// TIA Portal V15.1 export
// export: Created 2024-06-21T08:41:24.2160416Z, ExportSetting WithDefaults, DisplayName Totally Integrated Automation Portal, DisplayVersion V15.1 Update 5, DisplayName TIA Portal Openness, DisplayVersion V15.1 Update 5, DisplayName SINAMICS Startdrive Advanced, DisplayVersion V15.1, DisplayName G130, G150, S120, S150, SINAMICS MV, S210, DisplayVersion V15.1, DisplayName G110M, G120, G120C, G120D, G120P, DisplayVersion V15.1, DisplayName STEP 7 Professional, DisplayVersion V15.1 Update 5, DisplayName STEP 7 Safety, DisplayVersion V15.1, DisplayName WinCC Professional, DisplayVersion V15.1 Update 5, DisplayName SIMATIC Visualization Architect, DisplayVersion V15.1
FUNCTION "209210NCB02TagSequence" : Void   // FC341, FBD
TITLE = 209210NCB02TagSequence
{ S7_Optimized_Access := 'TRUE' }
AUTHOR : CSTAAL
VERSION : 0.1
// stored: AutoNumber false, IsIECCheckEnabled false, SetENOAutomatically False, UDAEnableTagReadback false
   VAR_OUTPUT
      O_AlarmA : Bool;   // Alarm A
      O_AlarmB : Bool;   // Alarm B
      O_AlarmC : Bool;   // Alarm C
      O_AlarmD : Bool;   // Alarm D
      O_AlarmABCondition : Bool;   // Alarms resetable
      H_IAnim : Word;   // Icon Animation
   END_VAR
BEGIN

REGION Network 1: **** 1 - Inputs **** HMI Commands
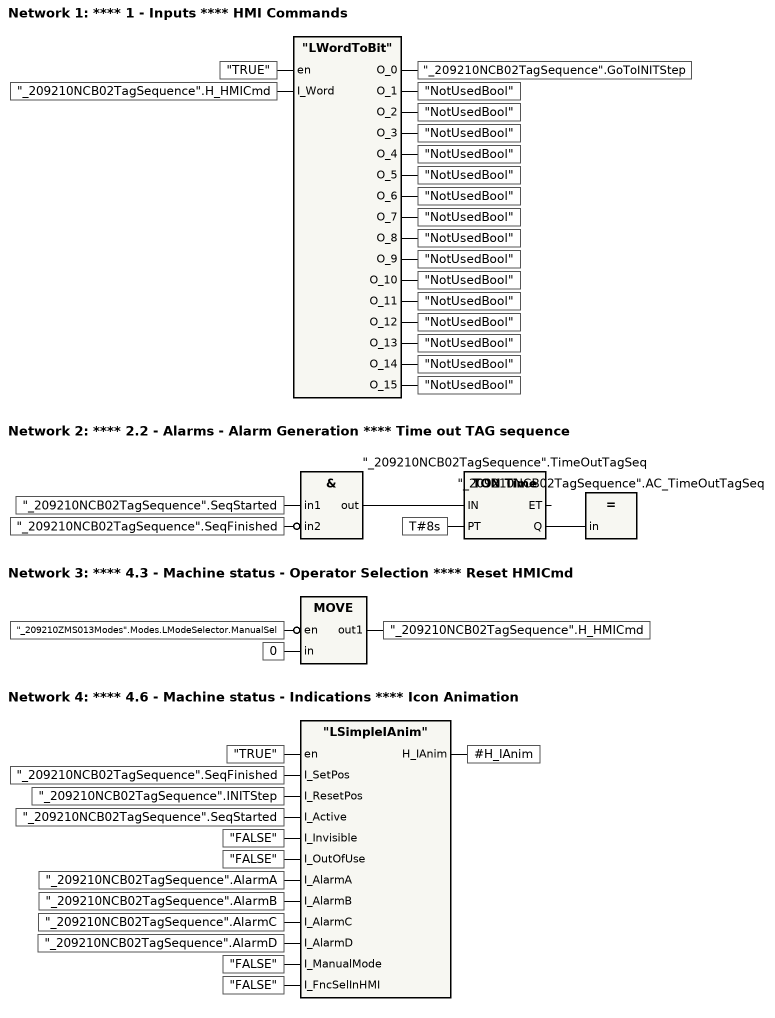
   IF "TRUE" THEN
       "LWordToBit"(I_Word := "_209210NCB02TagSequence".H_HMICmd,
                    O_0 => "_209210NCB02TagSequence".GoToINITStep,
                    O_1 => "NotUsedBool",
                    O_2 => "NotUsedBool",
                    O_3 => "NotUsedBool",
                    O_4 => "NotUsedBool",
                    O_5 => "NotUsedBool",
                    O_6 => "NotUsedBool",
                    O_7 => "NotUsedBool",
                    O_8 => "NotUsedBool",
                    O_9 => "NotUsedBool",
                    O_10 => "NotUsedBool",
                    O_11 => "NotUsedBool",
                    O_12 => "NotUsedBool",
                    O_13 => "NotUsedBool",
                    O_14 => "NotUsedBool",
                    O_15 => "NotUsedBool");
   END_IF;
END_REGION

REGION Network 2: **** 2.2 - Alarms - Alarm Generation **** Time out TAG sequence
   // Time out of the Tag Sequence
   "_209210NCB02TagSequence".TimeOutTagSeq.TON(IN := "_209210NCB02TagSequence".SeqStarted AND NOT "_209210NCB02TagSequence".SeqFinished,
                           PT := T#8s);
   "_209210NCB02TagSequence".AC_TimeOutTagSeq := "_209210NCB02TagSequence".TimeOutTagSeq.Q;
END_REGION

REGION Network 3: **** 4.3 - Machine status - Operator Selection **** Reset HMICmd
   // Reset HMICmd
   IF NOT "_209210ZMS013Modes".Modes.LModeSelector.ManualSel THEN
       "_209210NCB02TagSequence".H_HMICmd := 0;
   END_IF;
END_REGION

REGION Network 4: **** 4.6 - Machine status - Indications **** Icon Animation
   // Icon animation
   IF "TRUE" THEN
       "LSimpleIAnim"(I_SetPos := "_209210NCB02TagSequence".SeqFinished,
                      I_ResetPos := "_209210NCB02TagSequence".INITStep,
                      I_Active := "_209210NCB02TagSequence".SeqStarted,
                      I_Invisible := "FALSE",
                      I_OutOfUse := "FALSE",
                      I_AlarmA := "_209210NCB02TagSequence".AlarmA,
                      I_AlarmB := "_209210NCB02TagSequence".AlarmB,
                      I_AlarmC := "_209210NCB02TagSequence".AlarmC,
                      I_AlarmD := "_209210NCB02TagSequence".AlarmD,
                      I_ManualMode := "FALSE",
                      I_FncSelInHMI := "FALSE",
                      H_IAnim => #H_IAnim);
   END_IF;
END_REGION

REGION Network 5: **** 4.6 - Machine status - Indications **** Animation
   // Animation
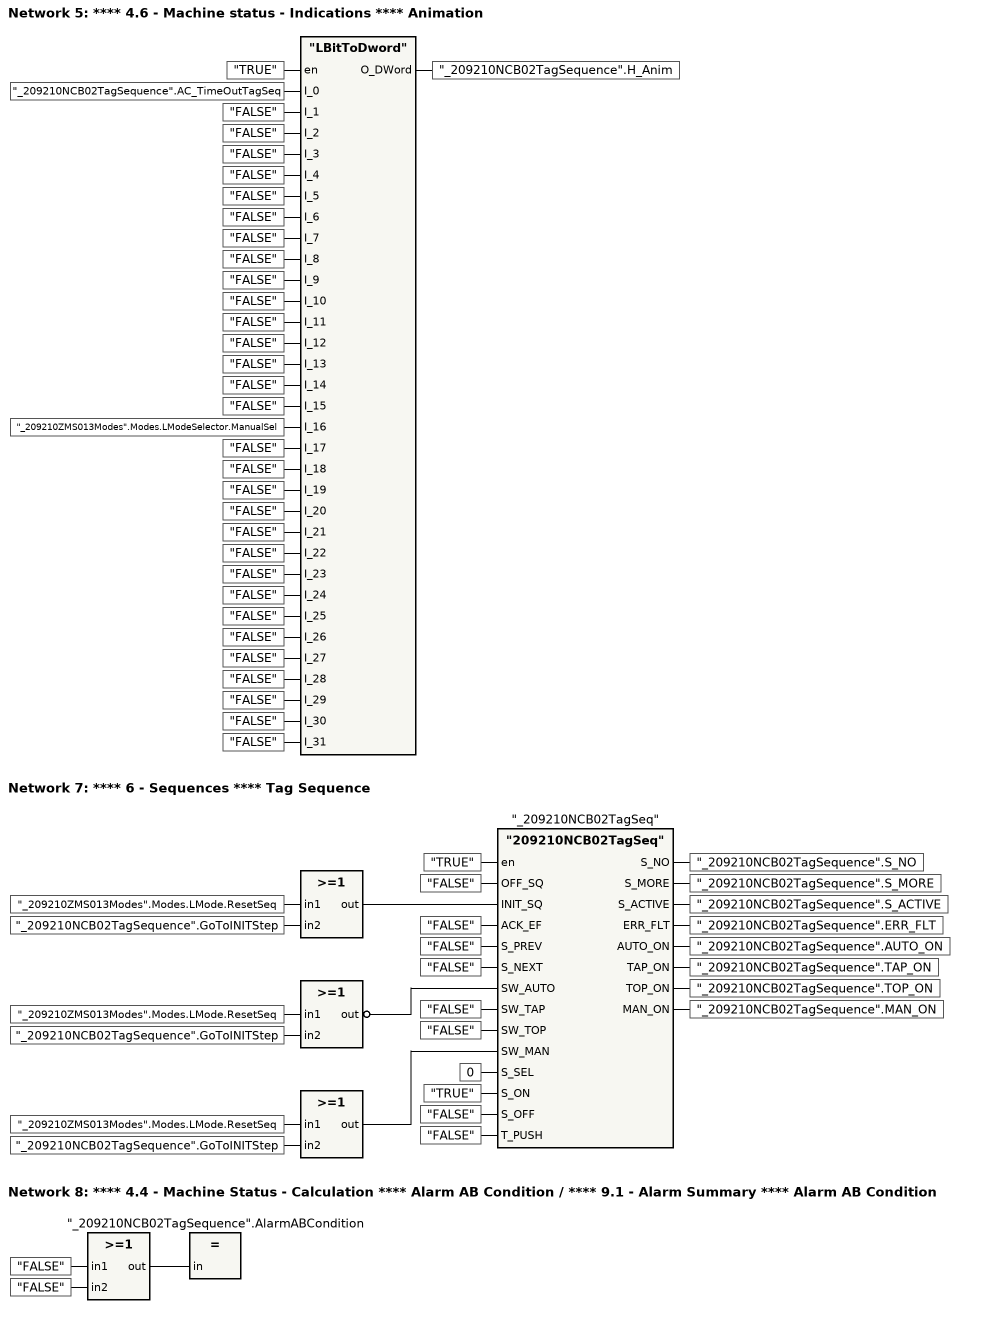
   IF "TRUE" THEN
       "LBitToDword"(I_0 := "_209210NCB02TagSequence".AC_TimeOutTagSeq,
                     I_1 := "FALSE",
                     I_2 := "FALSE",
                     I_3 := "FALSE",
                     I_4 := "FALSE",
                     I_5 := "FALSE",
                     I_6 := "FALSE",
                     I_7 := "FALSE",
                     I_8 := "FALSE",
                     I_9 := "FALSE",
                     I_10 := "FALSE",
                     I_11 := "FALSE",
                     I_12 := "FALSE",
                     I_13 := "FALSE",
                     I_14 := "FALSE",
                     I_15 := "FALSE",
                     I_16 := "_209210ZMS013Modes".Modes.LModeSelector.ManualSel,
                     I_17 := "FALSE",
                     I_18 := "FALSE",
                     I_19 := "FALSE",
                     I_20 := "FALSE",
                     I_21 := "FALSE",
                     I_22 := "FALSE",
                     I_23 := "FALSE",
                     I_24 := "FALSE",
                     I_25 := "FALSE",
                     I_26 := "FALSE",
                     I_27 := "FALSE",
                     I_28 := "FALSE",
                     I_29 := "FALSE",
                     I_30 := "FALSE",
                     I_31 := "FALSE",
                     O_DWord => "_209210NCB02TagSequence".H_Anim);
   END_IF;
END_REGION

NETWORK
TITLE = **** 4.6 - Machine Status - Indications **** Animation DB number
// DB number
      OPN   "_209210NCB02TagSequence";
      L     DBNO;
      T     "_209210NCB02TagSequence".H_DBnr;

REGION Network 7: **** 6 - Sequences **** Tag Sequence
   // Tag Sequence of the Antenna
   IF "TRUE" THEN
       "_209210NCB02TagSeq"(OFF_SQ := "FALSE",   // "209210NCB02TagSeq"
                            INIT_SQ := "_209210ZMS013Modes".Modes.LMode.ResetSeq OR "_209210NCB02TagSequence".GoToINITStep,
                            ACK_EF := "FALSE",
                            S_PREV := "FALSE",
                            S_NEXT := "FALSE",
                            SW_AUTO := NOT ("_209210ZMS013Modes".Modes.LMode.ResetSeq OR "_209210NCB02TagSequence".GoToINITStep),
                            SW_TAP := "FALSE",
                            SW_TOP := "FALSE",
                            SW_MAN := "_209210ZMS013Modes".Modes.LMode.ResetSeq OR "_209210NCB02TagSequence".GoToINITStep,
                            S_SEL := 0,
                            S_ON := "TRUE",
                            S_OFF := "FALSE",
                            T_PUSH := "FALSE",
                            S_NO => "_209210NCB02TagSequence".S_NO,
                            S_MORE => "_209210NCB02TagSequence".S_MORE,
                            S_ACTIVE => "_209210NCB02TagSequence".S_ACTIVE,
                            ERR_FLT => "_209210NCB02TagSequence".ERR_FLT,
                            AUTO_ON => "_209210NCB02TagSequence".AUTO_ON,
                            TAP_ON => "_209210NCB02TagSequence".TAP_ON,
                            TOP_ON => "_209210NCB02TagSequence".TOP_ON,
                            MAN_ON => "_209210NCB02TagSequence".MAN_ON);
   END_IF;
END_REGION

REGION Network 8: **** 4.4 - Machine Status - Calculation **** Alarm AB Condition / **** 9.1 - Alarm Summary **** Alarm AB Condition
   // Alarm AB Condition
   "_209210NCB02TagSequence".AlarmABCondition := "FALSE" OR "FALSE";
END_REGION

REGION Network 9: **** 9 - Alarm Summary **** Alarm A / **** 9.1 - Alarm Summary **** Alarm A
   // Upper level Alarm A
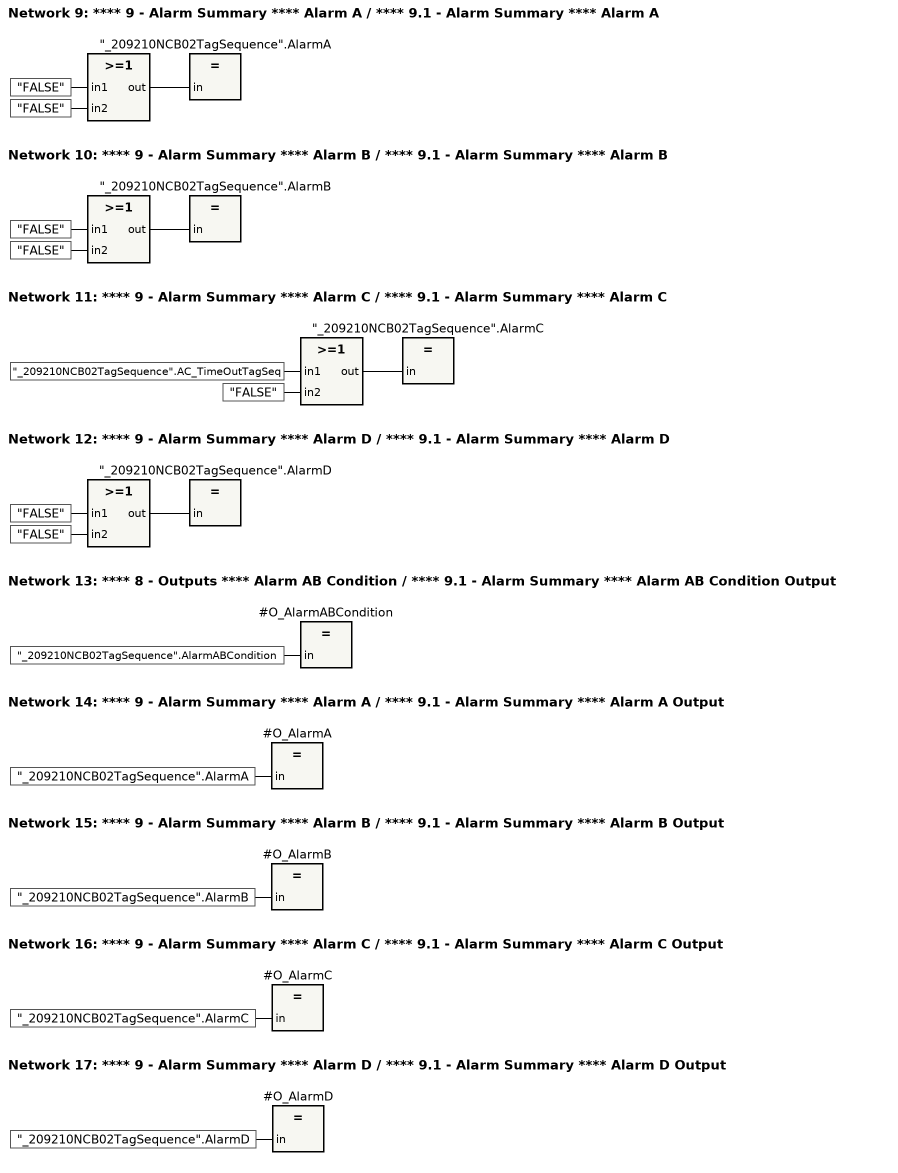
   "_209210NCB02TagSequence".AlarmA := "FALSE" OR "FALSE";
END_REGION

REGION Network 10: **** 9 - Alarm Summary **** Alarm B / **** 9.1 - Alarm Summary **** Alarm B
   // "_VV364".SZ1_AlarmUpper level Alarm B
   "_209210NCB02TagSequence".AlarmB := "FALSE" OR "FALSE";
END_REGION

REGION Network 11: **** 9 - Alarm Summary **** Alarm C / **** 9.1 - Alarm Summary **** Alarm C
   // Upper level Alarm B
   "_209210NCB02TagSequence".AlarmC := "_209210NCB02TagSequence".AC_TimeOutTagSeq OR "FALSE";
END_REGION

REGION Network 12: **** 9 - Alarm Summary **** Alarm D / **** 9.1 - Alarm Summary **** Alarm D
   // Upper level Alarm B
   "_209210NCB02TagSequence".AlarmD := "FALSE" OR "FALSE";
END_REGION

REGION Network 13: **** 8 - Outputs **** Alarm AB Condition / **** 9.1 - Alarm Summary **** Alarm AB Condition Output
   // Alarm AB Condition
   #O_AlarmABCondition := "_209210NCB02TagSequence".AlarmABCondition;
END_REGION

REGION Network 14: **** 9 - Alarm Summary **** Alarm A / **** 9.1 - Alarm Summary **** Alarm A Output
   // Upper level Alarm A
   #O_AlarmA := "_209210NCB02TagSequence".AlarmA;
END_REGION

REGION Network 15: **** 9 - Alarm Summary **** Alarm B / **** 9.1 - Alarm Summary **** Alarm B Output
   // "_VV364".SZ1_AlarmUpper level Alarm B
   #O_AlarmB := "_209210NCB02TagSequence".AlarmB;
END_REGION

REGION Network 16: **** 9 - Alarm Summary **** Alarm C / **** 9.1 - Alarm Summary **** Alarm C Output
   // Upper level Alarm B
   #O_AlarmC := "_209210NCB02TagSequence".AlarmC;
END_REGION

REGION Network 17: **** 9 - Alarm Summary **** Alarm D / **** 9.1 - Alarm Summary **** Alarm D Output
   // Upper level Alarm B
   #O_AlarmD := "_209210NCB02TagSequence".AlarmD;
END_REGION

REGION Network 18: **** 9.2 - Alarm DWord**** Alarm To DWord
   // Alarm Word
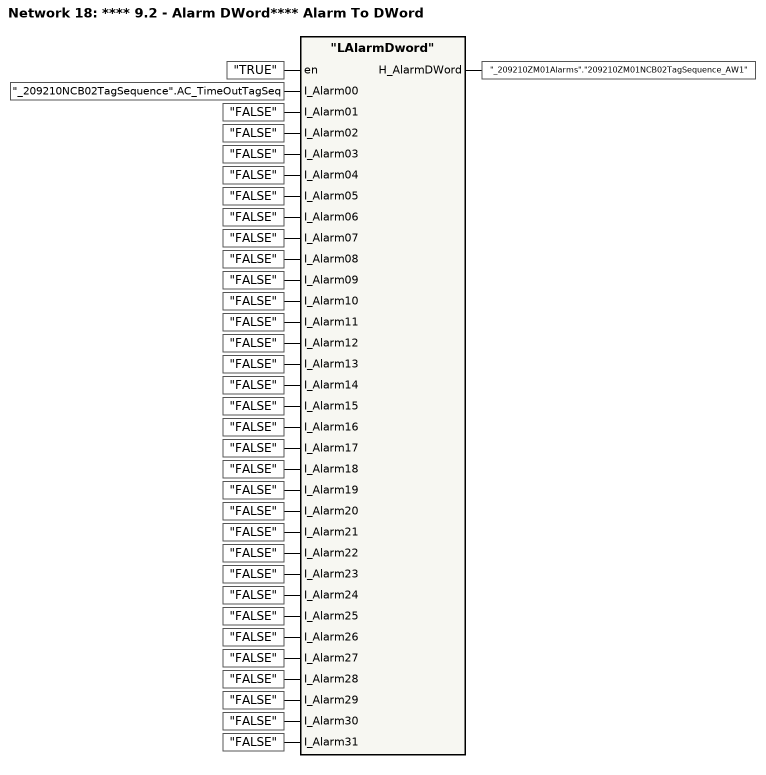
   IF "TRUE" THEN
       "LAlarmDword"(I_Alarm00 := "_209210NCB02TagSequence".AC_TimeOutTagSeq,
                     I_Alarm01 := "FALSE",
                     I_Alarm02 := "FALSE",
                     I_Alarm03 := "FALSE",
                     I_Alarm04 := "FALSE",
                     I_Alarm05 := "FALSE",
                     I_Alarm06 := "FALSE",
                     I_Alarm07 := "FALSE",
                     I_Alarm08 := "FALSE",
                     I_Alarm09 := "FALSE",
                     I_Alarm10 := "FALSE",
                     I_Alarm11 := "FALSE",
                     I_Alarm12 := "FALSE",
                     I_Alarm13 := "FALSE",
                     I_Alarm14 := "FALSE",
                     I_Alarm15 := "FALSE",
                     I_Alarm16 := "FALSE",
                     I_Alarm17 := "FALSE",
                     I_Alarm18 := "FALSE",
                     I_Alarm19 := "FALSE",
                     I_Alarm20 := "FALSE",
                     I_Alarm21 := "FALSE",
                     I_Alarm22 := "FALSE",
                     I_Alarm23 := "FALSE",
                     I_Alarm24 := "FALSE",
                     I_Alarm25 := "FALSE",
                     I_Alarm26 := "FALSE",
                     I_Alarm27 := "FALSE",
                     I_Alarm28 := "FALSE",
                     I_Alarm29 := "FALSE",
                     I_Alarm30 := "FALSE",
                     I_Alarm31 := "FALSE",
                     H_AlarmDWord => "_209210ZM01Alarms"."209210ZM01NCB02TagSequence_AW1");
   END_IF;
END_REGION
END_FUNCTION
